TYPE TcoMultiAxisStatus : STRUCT
    ActionDescription : STRING(100);
END_STRUCT
END_TYPE

(* stored: Version 1.1.0.1, ProductVersion 3.1.4024.12
   DUT TcoMultiAxisStatus: Id {8633d8a6-6ba1-09b2-261a-1d14e8315ecd} *)
